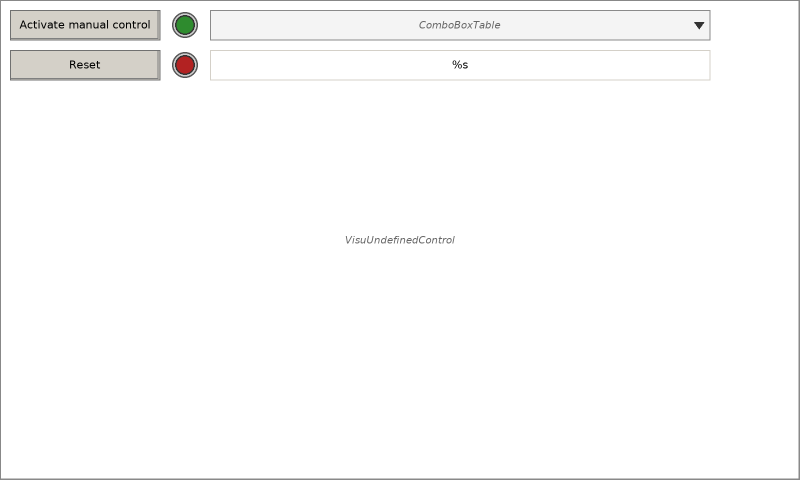
VISUALIZATION ManualControl  // 800x480
VAR_IN_OUT
	fbManualControler	: FB_ManualController ;
END_VAR
    Frame (0,0 800x480), input disabled if: fbManualControler.bDisableManualInputs, frame switch variable: fbManualControler.eDevType
        shows VisuUndefinedControl()
        shows VisuValveControl(fbManualControler := fbManualControler)
        shows VisuCylinderControl(fbManualControler := fbManualControler)
        shows VisuAxisControl(fbManualControler := fbManualControler)
        shows VisuPushbuttonLightControl(fbManualControler := fbManualControler)
        shows VisuDigitalInputControl(fbManualControler := fbManualControler)
        shows VisuAnlogInputControl(fbManualControler := fbManualControler)
        shows VisuDigitalOutControl(fbManualControler := fbManualControler)
        shows VisuAnalogOutControl(fbManualControler := fbManualControler)
        shows VisuPWMControl(fbManualControler := fbManualControler)
        shows VisuDoublePWMControl(fbManualControler := fbManualControler)
        shows VisuEncoderInput(fbManualControler := fbManualControler)
        shows VisuAnalogAxisControl(fbManualControler := fbManualControler)
        shows VisuTwoVelocityAxisControl(fbManualControler := fbManualControler)
        shows VisuKL5151Control(fbManualControler := fbManualControler)
        shows VisuKL15XXControl(fbManualControler := fbManualControler)
    Button (10,10 150x30), "Activate manual control", pressed state: fbManualControler.bManualActive
        toggle fbManualControler.bManualActive
    Lamp1 (170,50 30x30), tooltip "component fault active", variable: fbManualControler.bErroractive, style: Lamp-Lamp1-Red
    Lamp1 (170,10 30x30), tooltip "Manual control active", variable: fbManualControler.bManual, style: Lamp-Lamp1-Green
    Textfield (210,50 500x30), "%s", text variable: fbManualControler.sDeviceState
    Button (10,50 150x30), "Reset"
        tap fbManualControler.bReset
    ComboBoxTable (210,10 500x30), variable: fbManualControler.nCmdLookupindex, data array: fbManualControler.arDeviceArray
        p1128707560: fbManualControler.nNumberOfDevices
        p3854506369: fbManualControler.arDeviceArray[INDEX].sName
        p1892666644: fbManualControler.arDeviceArray[INDEX].sType
        p338671338: fbManualControler.arDeviceArray[INDEX].pFunction^
END_VISUALIZATION

(* stored: Version 1.1.0.1, ProductVersion 3.1.4024.11
   Visu ManualControl: Id {47fd7eab-4722-4161-bb7e-85fd17bf2676} *)
